// TIA Portal V20 export
TYPE "typeCmControlNodeInterlock"
// stored: Namespace Unit1.Em1
   STRUCT
      stacker2NgBoxLoading : "LER_typeTwoWayActuatorInterlock";
      stacker2NgBoxUnitMover : "LER_typeTwoWayActuatorInterlock";
      stacker2NgBoxClampLeft : "LER_typeTwoWayActuatorInterlock";
      stacker2NgBoxClampRight : "LER_typeTwoWayActuatorInterlock";
      stacker2NgBoxClampMover : "LER_typeTwoWayActuatorInterlock";
      stacker2NgBoxLift : "LER_typeTwoWayActuatorInterlock";
      stacker2NgBoxLock : "LER_typeTwoWayActuatorInterlock";
   END_STRUCT;
END_TYPE
